FUNCTION TryConvert_WORD_TO_LWORD : BOOL
VAR_INPUT
	in : WORD;
	out : REFERENCE TO LWORD;
END_VAR

out := WORD_TO_LWORD(in);
TryConvert_WORD_TO_LWORD := TRUE;

END_FUNCTION

(* stored: Version 1.1.0.1, ProductVersion 3.1.4024.12
   POU TryConvert_WORD_TO_LWORD: Id {5ba1c640-38b1-4fb3-9aac-93969113f9e5}, SpecialFunc None *)
